% RSLogix 500 project PID HEATER CONTROL.RSS, saved by version 8.30.00.16 %
PROJECT "UNTITLED"    % processor: Bul.1763 MicroLogix 1100 Series A %

PROGRAM FILES
  LAD 2   4 rungs

DATA FILES
  O0 OUTPUT  9 elements
  I1 INPUT  16 elements
  S2 STATUS  66 elements
  B3 BINARY  1 elements
  T4 TIMER  1 elements
  C5 COUNTER  1 elements
  R6 CONTROL  1 elements
  N7 INTEGER  2 elements
  F8 FLOAT  1 elements
  PD9 TEMP  1 elements

LADDER 2
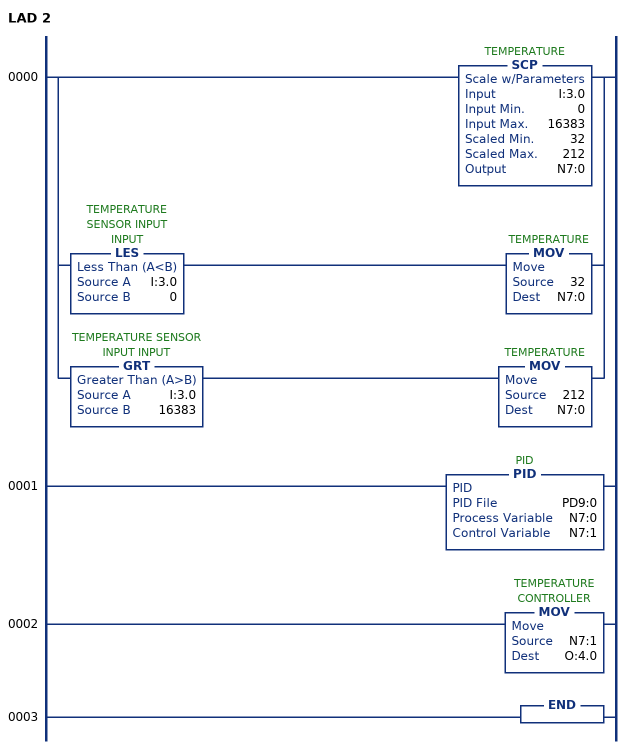
% Rung: 0 %
SOR BST BST SCP I:3.0 0 16383 32 212 N7:0 NXB LES I:3.0 0 MOV 32 N7:0 BND NXB GRT I:3.0 16383 MOV 212 N7:0 BND EOR
%   I:3.0  INPUT  "TEMPERATURE SENSOR INPUT" %
%   N7:0  "TEMPERATURE" %
% Rung: 1 %
SOR PID PD9:0 N7:0 N7:1 EOR
%   PD9:0  "PID" %
%   N7:0  "TEMPERATURE" %
%   N7:1  "PID OUTPUT" %
% Rung: 2 %
SOR MOV N7:1 O:4.0 EOR
%   N7:1  "PID OUTPUT" %
%   O:4.0  "TEMPERATURE CONTROLLER" %
% Rung: 3 %
SOR END EOR

OTHER DOCUMENTED ADDRESSES
  I:3.0/0  "TEMPERATURE SENSOR INPUT"
  O:4.0/0  "TEMPERATURE CONTROLLER"
